PROGRAM UpLimit
VAR	
	crush_left : ARRAY [1..5] OF WORD := [16#2A2A, 16#2A2A, 16#2A43, 16#5255, 16#5348];
	crush_right : ARRAY [1..5] OF WORD := [16#2046, 16#4155, 16#4C54, 16#2A2A, 16#2A2A];
	
	hard_left : ARRAY [1..5] OF WORD := [16#2A2A, 16#2A2A, 16#5550, 16#2048, 16#4152];
	hard_right : ARRAY [1..5] OF WORD := [16#4420, 16#4C49, 16#4D49, 16#542A, 16#2A2A];
	
	soft_left : ARRAY [1..5] OF WORD := [16#2A2A, 16#2A2A, 16#5550, 16#2053, 16#4F46];
	soft_right : ARRAY [1..5] OF WORD := [16#5420, 16#4C49, 16#4D49, 16#542A, 16#2A2A];	
	
	message_left : ARRAY [1..5] OF WORD := [16#2020, 16#504C, 16#4541, 16#5345, 16#204A];
	message_right : ARRAY [1..5] OF WORD := [16#4F47, 16#2044, 16#4F57, 16#4E20, 16#2020];
	
	current : ARRAY [1..5] OF WORD := [16#4375, 16#7272, 16#656E, 16#7420, 16#506F];
	pos : ARRAY [1..5] OF WORD := [16#7320, 16#2020, 16#2020, 16#2020, 16#2020];
	tick: INT := 0;
END_VAR

GV_MODBUS.twoLeft:= message_left;
GV_MODBUS.twoRight:= message_right;

IF GV_LIFT.CRUSH_PROTECTION_INDICATOR_OUT THEN
	GV_MODBUS.oneLeft := crush_left;
	GV_MODBUS.oneRight := crush_right;
ELSIF GV_LIFT.UP_LIMIT_INDICATOR_OUT THEN
	GV_MODBUS.oneLeft := hard_left;
	GV_MODBUS.oneRight := hard_right;
ELSIF GV_LIFT.CURRENT_POSITION > XML.savedvalues.UpSoftLim THEN
	GV_MODBUS.oneLeft := soft_left;
	GV_MODBUS.oneRight := soft_right;
END_IF

GV_MODBUS.threeLeft := GV_MODBUS.blank;
GV_MODBUS.threeRight := GV_MODBUS.blank;

GV_MODBUS.fourLeft:= current;
GV_MODBUS.fourRight:= GV_MODBUS.blank;	

GV_MODBUS.fourRight:= Position_To_Row_Array(pos, GV_LIFT.CURRENT_POSITION);     


IF tick >= GV_MODBUS.refreshInterval THEN
	Execute_Write_Screen();
	tick := 0;
END_IF

tick := tick + 1;

END_PROGRAM

(* stored: Version 1.1.0.1, ProductVersion 3.1.4022.12
   POU UpLimit: Id {e6866071-58cb-426d-9411-09cfc3e0f235}, SpecialFunc None *)
